# EPICS substitutions: mc07/tpmacApp/Db/autohome.substitutions
file "db/autohome.db"
{
pattern
{SYS,                  DEV,                   PLC,  PORT  }
{"XF:16IDC-OP",        "{Slt:DDA-Ax:X}",      8,    P0    }
{"XF:16IDC-OP",        "{Slt:DDA-Ax:Y}",      9,    P0    }
{"XF:16IDC-OP",        "{Slt:DDA-Ax:dX}",     10,   P0    }
{"XF:16IDC-OP",        "{Slt:DDA-Ax:dY}",     11,   P0    }
{"XF:16IDC-ES:InAir",  "{Mscp:1-Ax:Pol}",    12,   P0    }
}
